(* Logix 5000 project; controller LADDER_APM_1 Emulate 5570 rev 32.11; software revision 32.00 *)

TASK MainTask (continuous, watchdog 500 ms) : MainProgram

MODULES
   Local : Emulate 5570 (ICP 2, rev 32.11)
      IN_OUT : vendor 1 type 0 code 15 (ICP 4, rev 1.1, Output RPI 5 ms)
END_MODULES

TYPE Drivers_CortadoraZ :
STRUCT
   MAM_CortadoraZ : MOTION_INSTRUCTION[3];
   MAS_CortadoraZ : MOTION_INSTRUCTION[3];
   MAH_CortadoraZ : MOTION_INSTRUCTION;
   MAJ_CortadoraZ : MOTION_INSTRUCTION;
END_STRUCT
END_TYPE

TYPE Drivers_Grupo :
STRUCT
   MGSD : MOTION_INSTRUCTION;
   MGS : MOTION_INSTRUCTION;
   MAFR : MOTION_INSTRUCTION;
   MASR : MOTION_INSTRUCTION;
   MGSR : MOTION_INSTRUCTION;
END_STRUCT
END_TYPE

TYPE Drivers_Mordaza :
STRUCT
   MAM_Mordaza : MOTION_INSTRUCTION[3];
   MAS_Mordaza : MOTION_INSTRUCTION[3];
   MAH_Mordaza : MOTION_INSTRUCTION;
   MAJ_Mordaza : MOTION_INSTRUCTION;
END_STRUCT
END_TYPE

VAR_GLOBAL   (* controller tags *)
   Driver_Grupo : Drivers_Grupo;
   Eje_CortadoraZ : AXIS_VIRTUAL;
   Eje_CortadoraZ_d : Drivers_CortadoraZ := (MAM_CortadoraZ[0].FLAGS := 704643072, MAM_CortadoraZ[0].DN := 1, MAM_CortadoraZ[0].PC := 1, MAM_CortadoraZ[1].FLAGS := 704643072, MAM_CortadoraZ[1].DN := 1, MAM_CortadoraZ[1].PC := 1);
   Eje_Mordaza : AXIS_VIRTUAL;
   Eje_Mordaza_d : Drivers_Mordaza := (MAM_Mordaza[0].FLAGS := 704643072, MAM_Mordaza[0].DN := 1, MAM_Mordaza[0].PC := 1, MAM_Mordaza[1].FLAGS := 704643072, MAM_Mordaza[1].DN := 1, MAM_Mordaza[1].PC := 1);
   Ejes_virtuales : MOTION_GROUP;
   Posicion_Cortadora : REAL;
   Posicion_Mordaza : REAL;
   PRUEBA : BOOL;
END_VAR

PROGRAM MainProgram   (* main routine MainRoutine *)
VAR
   BE : BOOL;
   BLP1 : BOOL;
   BLP2 : BOOL;
   BLP3 : BOOL;
   BS : BOOL := 1;
   DC : BOOL;
   DCA : BOOL;
   DCD : BOOL;
   LP : DINT;
   M : BOOL;
   MA : BOOL := 1;
   MARCHA : BOOL;
   MC : BOOL;
   PARADA : BOOL;
   Q0 : BOOL;
   Q1 : BOOL;
   Q10 : BOOL := 1;
   Q2 : BOOL;
   Q3 : BOOL;
   Q4 : BOOL;
   Q5 : BOOL;
   Q6 : BOOL;
   Q7 : BOOL;
   Q8 : BOOL;
   Q9 : BOOL;
   SC1 : BOOL;
   SC2 : BOOL;
   SC3 : BOOL;
   T_DCA : TIMER := (PRE := 6000);
   T_DCD : TIMER := (PRE := 6000);
   T_MA : TIMER := (PRE := 3000);
   T_MC : TIMER := (PRE := 3000, EN := 1, TT := 1);
   T_ZCA : TIMER := (PRE := 3000);
   T_ZCB : TIMER := (PRE := 3000);
   ZC_mas : BOOL;
   ZC_menos : BOOL;
   ZCA : BOOL := 1;
   ZCB : BOOL;
END_VAR

ROUTINE COMBINACIONAL   (* ladder *)
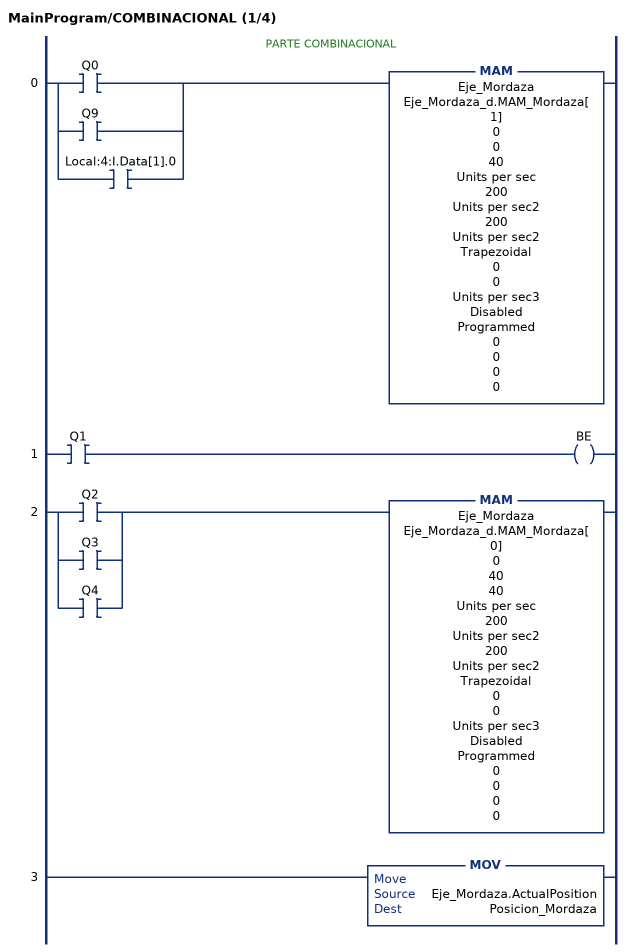
   // PARTE COMBINACIONAL
   0: [XIC(Q0) ,[XIC(Q9) ,XIC(Local:4:I.Data[1].0) ] ]MAM(Eje_Mordaza,Eje_Mordaza_d.MAM_Mordaza[1],0,0,40,Units per sec,200,Units per sec2,200,Units per sec2,Trapezoidal,0,0,Units per sec3,Disabled,Programmed,0,0,0,0);
   1: XIC(Q1)OTE(BE);
   2: [XIC(Q2) ,[XIC(Q3) ,XIC(Q4) ] ]MAM(Eje_Mordaza,Eje_Mordaza_d.MAM_Mordaza[0],0,40,40,Units per sec,200,Units per sec2,200,Units per sec2,Trapezoidal,0,0,Units per sec3,Disabled,Programmed,0,0,0,0);
   3: MOV(Eje_Mordaza.ActualPosition,Posicion_Mordaza);
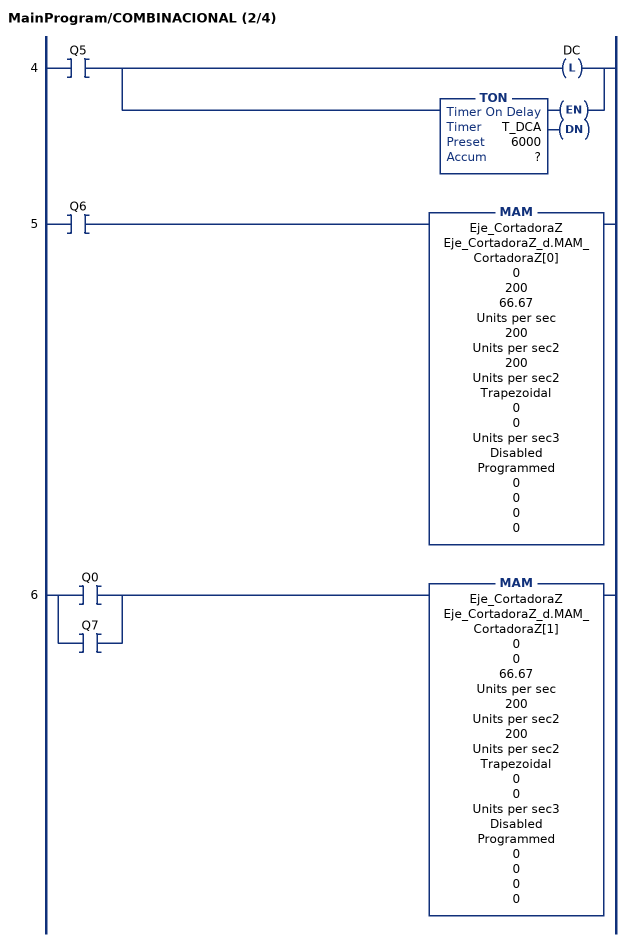
   4: XIC(Q5)[OTL(DC) ,TON(T_DCA,?,?) ];
   5: XIC(Q6)MAM(Eje_CortadoraZ,Eje_CortadoraZ_d.MAM_CortadoraZ[0],0,200,66.67,Units per sec,200,Units per sec2,200,Units per sec2,Trapezoidal,0,0,Units per sec3,Disabled,Programmed,0,0,0,0);
   6: [XIC(Q0) ,XIC(Q7) ]MAM(Eje_CortadoraZ,Eje_CortadoraZ_d.MAM_CortadoraZ[1],0,0,66.67,Units per sec,200,Units per sec2,200,Units per sec2,Trapezoidal,0,0,Units per sec3,Disabled,Programmed,0,0,0,0);
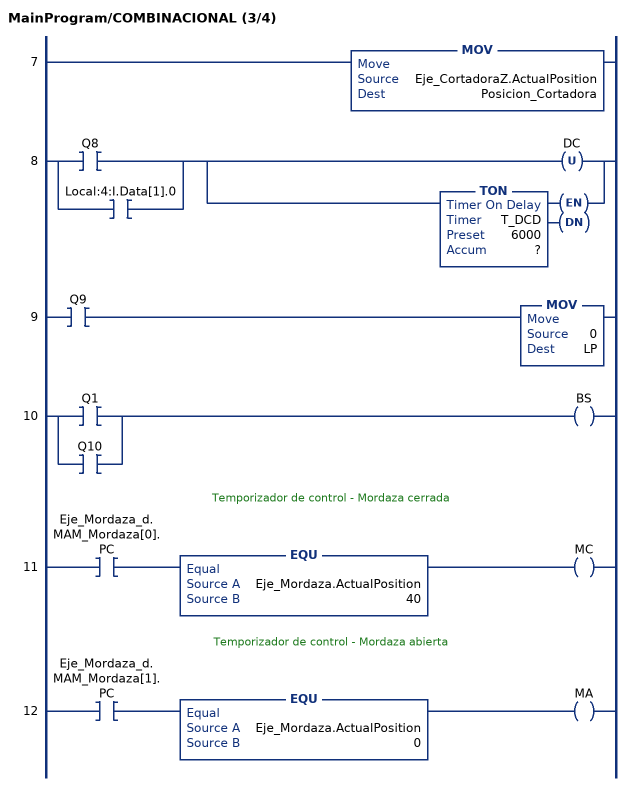
   7: MOV(Eje_CortadoraZ.ActualPosition,Posicion_Cortadora);
   8: [XIC(Q8) ,XIC(Local:4:I.Data[1].0) ][OTU(DC) ,TON(T_DCD,?,?) ];
   9: XIC(Q9)MOV(0,LP);
   10: [XIC(Q1) ,XIC(Q10) ]OTE(BS);
   // Temporizador de control - Mordaza cerrada
   11: XIC(Eje_Mordaza_d.MAM_Mordaza[0].PC)EQU(Eje_Mordaza.ActualPosition,40)OTE(MC);
   // Temporizador de control - Mordaza abierta
   12: XIC(Eje_Mordaza_d.MAM_Mordaza[1].PC)EQU(Eje_Mordaza.ActualPosition,0)OTE(MA);
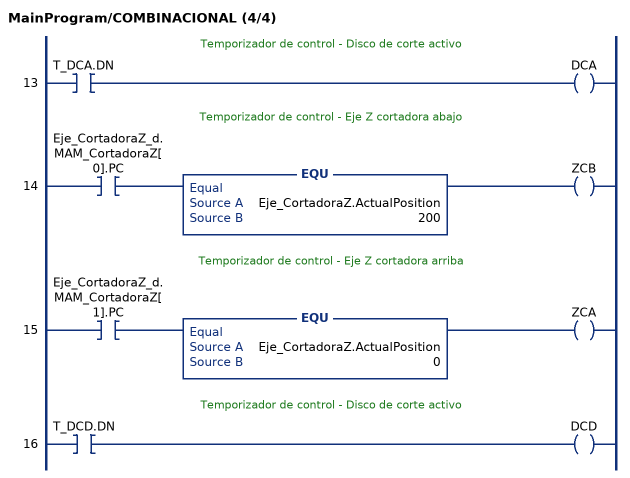
   // Temporizador de control - Disco de corte activo
   13: XIC(T_DCA.DN)OTE(DCA);
   // Temporizador de control - Eje Z cortadora abajo
   14: XIC(Eje_CortadoraZ_d.MAM_CortadoraZ[0].PC)EQU(Eje_CortadoraZ.ActualPosition,200)OTE(ZCB);
   // Temporizador de control - Eje Z cortadora arriba
   15: XIC(Eje_CortadoraZ_d.MAM_CortadoraZ[1].PC)EQU(Eje_CortadoraZ.ActualPosition,0)OTE(ZCA);
   // Temporizador de control - Disco de corte activo
   16: XIC(T_DCD.DN)OTE(DCD);
END_ROUTINE

ROUTINE MainRoutine   (* ladder *)
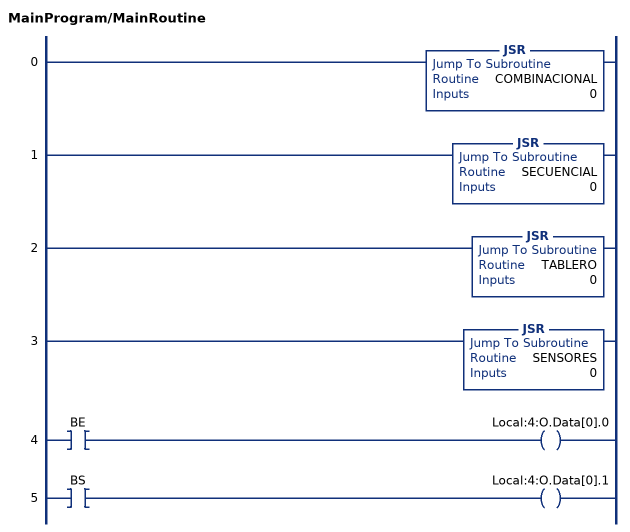
   0: JSR(COMBINACIONAL,0);
   1: JSR(SECUENCIAL,0);
   2: JSR(TABLERO,0);
   3: JSR(SENSORES,0);
   4: XIC(BE)OTE(Local:4:O.Data[0].0);
   5: XIC(BS)OTE(Local:4:O.Data[0].1);
END_ROUTINE

ROUTINE SECUENCIAL   (* ladder *)
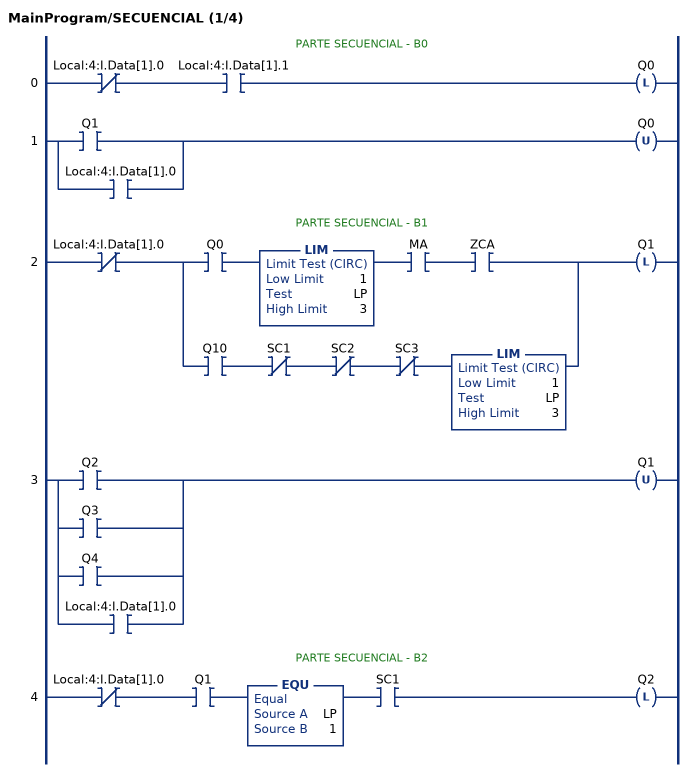
   // PARTE SECUENCIAL - B0
   0: XIO(Local:4:I.Data[1].0)XIC(Local:4:I.Data[1].1)OTL(Q0);
   1: [XIC(Q1) ,XIC(Local:4:I.Data[1].0) ]OTU(Q0);
   // PARTE SECUENCIAL - B1
   2: XIO(Local:4:I.Data[1].0)[XIC(Q0) LIM(1,LP,3) XIC(MA) XIC(ZCA) ,XIC(Q10) XIO(SC1) XIO(SC2) XIO(SC3) LIM(1,LP,3) ]OTL(Q1);
   3: [XIC(Q2) ,[XIC(Q3) ,[XIC(Q4) ,XIC(Local:4:I.Data[1].0) ] ] ]OTU(Q1);
   // PARTE SECUENCIAL - B2
   4: XIO(Local:4:I.Data[1].0)XIC(Q1)EQU(LP,1)XIC(SC1)OTL(Q2);
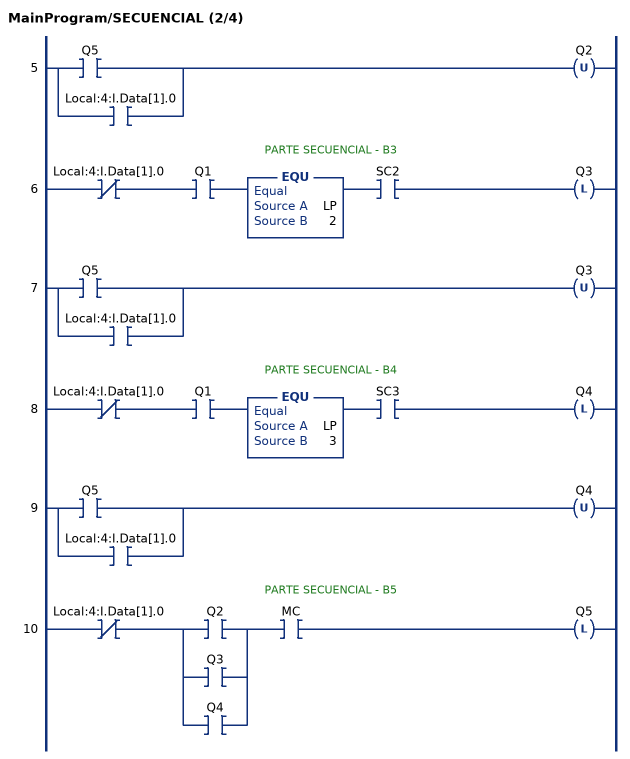
   5: [XIC(Q5) ,XIC(Local:4:I.Data[1].0) ]OTU(Q2);
   // PARTE SECUENCIAL - B3
   6: XIO(Local:4:I.Data[1].0)XIC(Q1)EQU(LP,2)XIC(SC2)OTL(Q3);
   7: [XIC(Q5) ,XIC(Local:4:I.Data[1].0) ]OTU(Q3);
   // PARTE SECUENCIAL - B4
   8: XIO(Local:4:I.Data[1].0)XIC(Q1)EQU(LP,3)XIC(SC3)OTL(Q4);
   9: [XIC(Q5) ,XIC(Local:4:I.Data[1].0) ]OTU(Q4);
   // PARTE SECUENCIAL - B5
   10: XIO(Local:4:I.Data[1].0)[XIC(Q2) ,[XIC(Q3) ,XIC(Q4) ] ]XIC(MC)OTL(Q5);
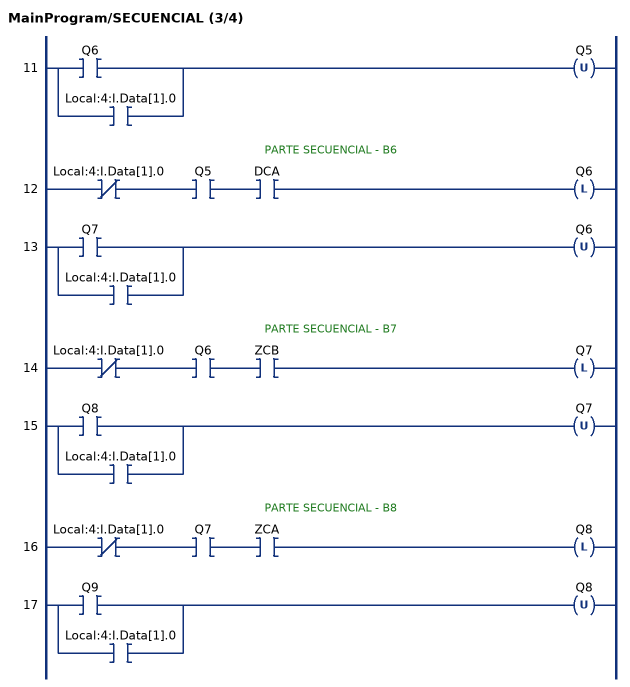
   11: [XIC(Q6) ,XIC(Local:4:I.Data[1].0) ]OTU(Q5);
   // PARTE SECUENCIAL - B6
   12: XIO(Local:4:I.Data[1].0)XIC(Q5)XIC(DCA)OTL(Q6);
   13: [XIC(Q7) ,XIC(Local:4:I.Data[1].0) ]OTU(Q6);
   // PARTE SECUENCIAL - B7
   14: XIO(Local:4:I.Data[1].0)XIC(Q6)XIC(ZCB)OTL(Q7);
   15: [XIC(Q8) ,XIC(Local:4:I.Data[1].0) ]OTU(Q7);
   // PARTE SECUENCIAL - B8
   16: XIO(Local:4:I.Data[1].0)XIC(Q7)XIC(ZCA)OTL(Q8);
   17: [XIC(Q9) ,XIC(Local:4:I.Data[1].0) ]OTU(Q8);
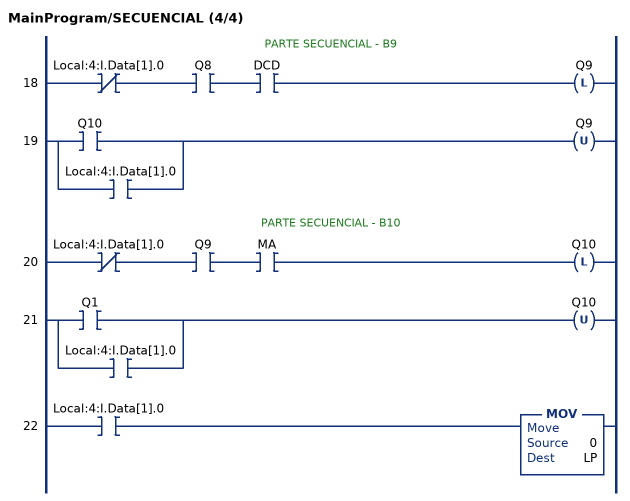
   // PARTE SECUENCIAL - B9
   18: XIO(Local:4:I.Data[1].0)XIC(Q8)XIC(DCD)OTL(Q9);
   19: [XIC(Q10) ,XIC(Local:4:I.Data[1].0) ]OTU(Q9);
   // PARTE SECUENCIAL - B10
   20: XIO(Local:4:I.Data[1].0)XIC(Q9)XIC(MA)OTL(Q10);
   21: [XIC(Q1) ,XIC(Local:4:I.Data[1].0) ]OTU(Q10);
   22: XIC(Local:4:I.Data[1].0)MOV(0,LP);
END_ROUTINE

ROUTINE SENSORES   (* ladder *)
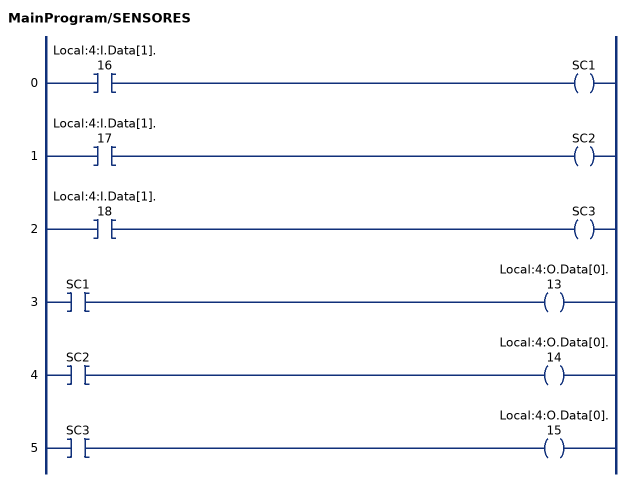
   0: XIC(Local:4:I.Data[1].16)OTE(SC1);
   1: XIC(Local:4:I.Data[1].17)OTE(SC2);
   2: XIC(Local:4:I.Data[1].18)OTE(SC3);
   3: XIC(SC1)OTE(Local:4:O.Data[0].13);
   4: XIC(SC2)OTE(Local:4:O.Data[0].14);
   5: XIC(SC3)OTE(Local:4:O.Data[0].15);
END_ROUTINE

ROUTINE TABLERO   (* ladder *)
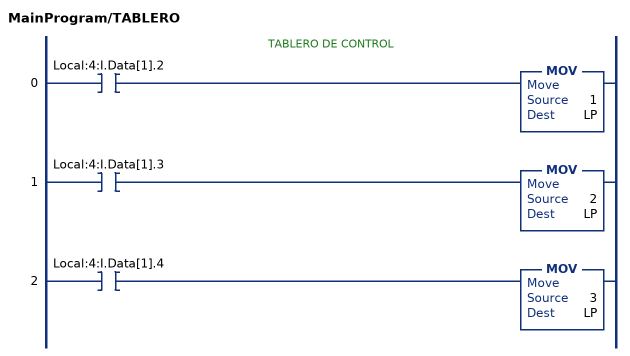
   // TABLERO DE CONTROL
   0: XIC(Local:4:I.Data[1].2)MOV(1,LP);
   1: XIC(Local:4:I.Data[1].3)MOV(2,LP);
   2: XIC(Local:4:I.Data[1].4)MOV(3,LP);
END_ROUTINE
END_PROGRAM
